Fanuc KAREL source: SEND_DATAPC.kl

PROGRAM T
%NOLOCKGROUP
VAR
 v0 : INTEGER
 v1 : ARRAY[20] OF BYTE
 v2 : INTEGER
BEGIN
 SEND_DATAPC(v0, v1, v2)
END T
